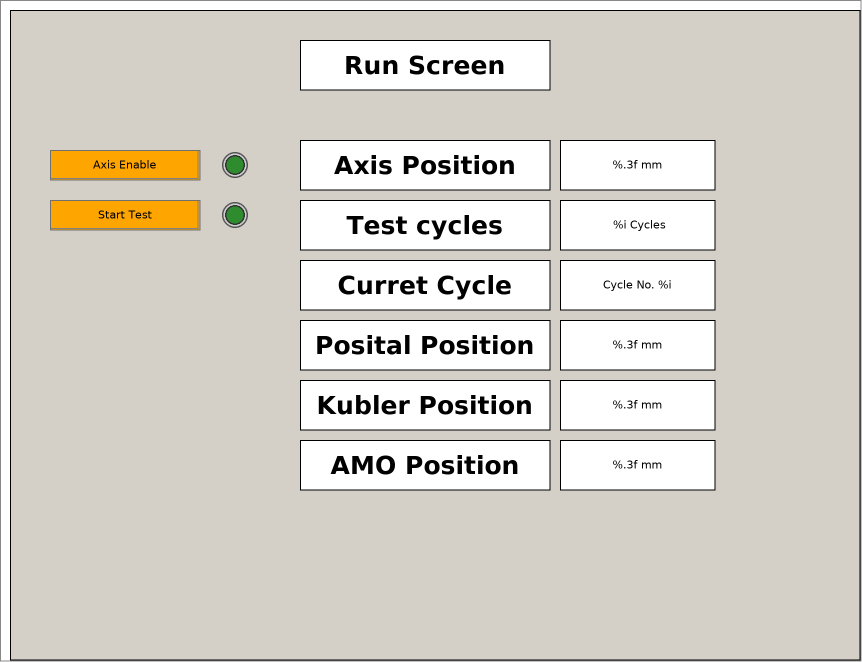
VISUALIZATION Run_Screen  // 862x662
    RoundedRectangle (10,10 850x650)
    RoundedRectangle (300,40 250x50), "Run Screen"
    Button (50,150 150x30), "Axis Enable"
        toggle MAIN.bEnableAxis_1
    Lamp1 (220,150 30x30), variable: MAIN.mcPower_1.Enable, style: Lamp-Lamp1-Green
    RoundedRectangle (300,140 250x50), "Axis Position"
    RoundedRectangle (560,140 155x50), "%.3f mm", text variable: GVL.stAxis_1.NcToPlc.SetPos
    RoundedRectangle (300,200 250x50), "Test cycles"
    RoundedRectangle (300,260 250x50), "Curret Cycle"
    RoundedRectangle (560,200 155x50), "%i Cycles", text variable: MAIN.fbTestCycleCounter.PV
    RoundedRectangle (560,260 155x50), "Cycle No. %i", text variable: MAIN.fbTestCycleCounter.CV
    Button (50,200 150x30), "Start Test"
        toggle MAIN.bStartTest
    Lamp1 (220,200 30x30), variable: MAIN.bStartTest, style: Lamp-Lamp1-Green
    RoundedRectangle (300,440 250x50), "AMO Position"
    RoundedRectangle (300,380 250x50), "Kubler Position"
    RoundedRectangle (300,320 250x50), "Posital Position"
    RoundedRectangle (560,380 155x50), "%.3f mm", text variable: stAxis_3.NcToPlc.ActPos
    RoundedRectangle (560,440 155x50), "%.3f mm", text variable: stAxis_4.NcToPlc.ActPos
    RoundedRectangle (560,320 155x50), "%.3f mm", text variable: stAxis_2.NcToPlc.ActPos
END_VISUALIZATION

(* stored: Version 1.1.0.1, ProductVersion 3.1.4024.0
   Visu Run_Screen: Id {6b199cb4-1a8f-4159-b339-5a9a860145f9} *)
